# EPICS autosave request: electronAnalyserViewerApp/Db/commonPlugin_noMagick_settings.req
file "NDPluginBase_settings.req",   P=$(P),  R=netCDF1:
file "NDFile_settings.req",         P=$(P),  R=netCDF1:
file "NDPluginBase_settings.req",   P=$(P),  R=TIFF1:
file "NDFile_settings.req",         P=$(P),  R=TIFF1:
file "NDPluginBase_settings.req",   P=$(P),  R=JPEG1:
file "NDFile_settings.req",         P=$(P),  R=JPEG1:
file "NDFileJPEG_settings.req",     P=$(P),  R=JPEG1:
file "NDPluginBase_settings.req",   P=$(P),  R=Nexus1:
file "NDFile_settings.req",         P=$(P),  R=Nexus1:
file "NDFileNexus_settings.req",    P=$(P),  R=Nexus1:
#!file "NDPluginBase_settings.req",   P=$(P),  R=Magick1:
#!file "NDFile_settings.req",         P=$(P),  R=Magick1:
#!file "NDFileMagick_settings.req",   P=$(P),  R=Magick1:
file "NDPluginBase_settings.req",   P=$(P),  R=HDF1:
file "NDFile_settings.req",         P=$(P),  R=HDF1:
file "NDFileHDF5_settings.req",      P=$(P),  R=HDF1:
file "NDPluginBase_settings.req",   P=$(P),  R=ROI1:
file "NDROI_settings.req",          P=$(P),  R=ROI1:
file "NDPluginBase_settings.req",   P=$(P),  R=ROI2:
file "NDROI_settings.req",          P=$(P),  R=ROI2:
file "NDPluginBase_settings.req",   P=$(P),  R=ROI3:
file "NDROI_settings.req",          P=$(P),  R=ROI3:
file "NDPluginBase_settings.req",   P=$(P),  R=ROI4:
file "NDROI_settings.req",          P=$(P),  R=ROI4:
file "NDPluginBase_settings.req",   P=$(P),  R=Proc1:
file "NDProcess_settings.req",      P=$(P),  R=Proc1:
file "NDPluginBase_settings.req",   P=$(P),  R=Stats1:
file "NDStats_settings.req",        P=$(P),  R=Stats1:
file "NDPluginBase_settings.req",   P=$(P),  R=Stats2:
file "NDStats_settings.req",        P=$(P),  R=Stats2:
file "NDPluginBase_settings.req",   P=$(P),  R=Stats3:
file "NDStats_settings.req",        P=$(P),  R=Stats3:
file "NDPluginBase_settings.req",   P=$(P),  R=Stats4:
file "NDStats_settings.req",        P=$(P),  R=Stats4:
file "NDPluginBase_settings.req",   P=$(P),  R=Stats5:
file "NDStats_settings.req",        P=$(P),  R=Stats5:
file "NDPluginBase_settings.req",   P=$(P),  R=Trans1:
file "NDTransform_settings.req",    P=$(P),  R=Trans1:
file "NDPluginBase_settings.req",   P=$(P),  R=Over1:
file "NDOverlay_settings.req",      P=$(P),  R=Over1:
file "NDOverlayN_settings.req",     P=$(P),  R=Over1:1:
file "NDOverlayN_settings.req",     P=$(P),  R=Over1:2:
file "NDOverlayN_settings.req",     P=$(P),  R=Over1:3:
file "NDOverlayN_settings.req",     P=$(P),  R=Over1:4:
file "NDOverlayN_settings.req",     P=$(P),  R=Over1:5:
file "NDOverlayN_settings.req",     P=$(P),  R=Over1:6:
file "NDOverlayN_settings.req",     P=$(P),  R=Over1:7:
file "NDOverlayN_settings.req",     P=$(P),  R=Over1:8:
file "NDPluginBase_settings.req",   P=$(P),  R=CC1:
file "NDColorConvert_settings.req", P=$(P),  R=CC1:
file "NDPluginBase_settings.req",   P=$(P),  R=CC2:
file "NDColorConvert_settings.req", P=$(P),  R=CC2:
file "scan_settings.req",           P=$(P),  S=scan1
file "scan_settings.req",           P=$(P),  S=scan2
file "scan_settings.req",           P=$(P),  S=scan3
file "scan_settings.req",           P=$(P),  S=scan4
file "sseq_settings.req",           P=$(P),  S=AcquireSequence
